// TIA Portal V19 export
FUNCTION_BLOCK "CameraConnectionTCP"   // FB2, LAD
{ S7_Optimized_Access := 'TRUE' }
// stored: MemoryReserve 100, SetENOAutomatically false
   VAR_INPUT
      Enable : Bool;
      Execute : Bool;
      Reset : Bool;
      ConnectionTimer : Time;
   END_VAR
   VAR_OUTPUT
      Status : "Status";
   END_VAR
   VAR_IN_OUT
      Parameters : TCON_IP_v4;
   END_VAR
   VAR
      TCON_Instance { ExternalAccessible := 'False'; ExternalVisible := 'False'; ExternalWritable := 'False'} : TCON;
      TDISCON_Instance { ExternalAccessible := 'False'; ExternalVisible := 'False'; ExternalWritable := 'False'} : TDISCON;
      TRCV_Instance { ExternalAccessible := 'False'; ExternalVisible := 'False'; ExternalWritable := 'False'} : TRCV;
      TSEND_Instance { ExternalAccessible := 'False'; ExternalVisible := 'False'; ExternalWritable := 'False'} : TSEND;
      Connection : Struct
         TCON : Struct
            REQ : Bool;
            BUSY : Bool;
            DONE : Bool;
            ERROR : Bool;
            STATUS : Word;
            CONNECTION_DATA : Struct
               InterfaceID : HW_ANY := 64;
               ID : HW_ANY := 1;
               ConnectionType : Byte := 16#0B;
               ActiveEstablished : Bool := false;
               RemodeAddress { S7_SetPoint := 'True'} : IP_V4;
               RemotePort : UInt;
               LocalPort : UInt := 2000;
            END_STRUCT;
         END_STRUCT;
         TDISCON : Struct
            REQ : Bool;
            BUSY : Bool;
            DONE : Bool;
            ERROR : Bool;
            STATUS : Word;
         END_STRUCT;
         TSEND : Struct
            REQ : Bool;
            LEN : UDInt;
            BUSY : Bool;
            DONE : Bool;
            ERROR : Bool;
            STATUS : Word;
         END_STRUCT;
         TRVC : Struct
            ENABLE : Bool;
            ADHOC : Bool := TRUE;
            LEN : UDInt;
            NDR : Bool;
            BUSY : Bool;
            RVC_LEN : UDInt;
            ERROR : Bool;
            STATUS : Word;
         END_STRUCT;
      END_STRUCT;
      Data : Struct
         RVC : Array[0..999] of Byte;
         SEND : Array[0..999] of Byte;
      END_STRUCT;
      State : "s_changeState";
      Timers : Struct
         WatchdogInit : "s_TON";
         WatchdogCamera : "s_TON";
         WatchdogInitRVC { S7_SetPoint := 'True'} : "s_TON";
         WatchdogMachineStart { S7_SetPoint := 'True'} : "s_TON";
      END_STRUCT;
      MessageGenerating : Struct
         i : Int;
         len : DInt;
         "string" : String[100];
         chars : Array[0..99] of Char;
      END_STRUCT;
      Local : Struct
         MessageSent : Bool;
         MessageSentCounter : SInt;
         prevState : Int;
      END_STRUCT;
      F_TRIG_Enable { ExternalAccessible := 'False'; ExternalVisible := 'False'; ExternalWritable := 'False'} : F_TRIG;
      R_TRIG_Execute { ExternalAccessible := 'False'; ExternalVisible := 'False'; ExternalWritable := 'False'} : R_TRIG;
      R_TRIG_Enable { ExternalAccessible := 'False'; ExternalVisible := 'False'; ExternalWritable := 'False'} : R_TRIG;
      Connected : Bool;
      DebugCounter : DInt;
   END_VAR
   VAR CONSTANT
      S_INITIALIZE : Int := 1;
      S_DISCONNECT : Int := 10;
      S_ERROR : Int := 20;
      S_ENABLE_RVC : Int := 30;
      S_MACHINE_START : Int := 40;
      S_IDLE : Int := 50;
      S_START_CAMERA : Int := 60;
      S_REPEAT : Int := 70;
      STATE_TEST : Int := 100;
      COMAND_SEND_MACHINE_START : String := 'command: machine_start';
      COMMAND_RVC_MACHINE_START : String := 'command: camera_ready';
      COMMAND_SEND_START_CONTROL : String := 'command: start_control';
      COMMAND_RVC_CONTROL_DONE : String := 'command: control_done';
      E_CONNECTION_TIMEOUT : Word := 16#8000;
      E_WRONG_RESPONSE_MACHINE_START : Word := 16#8001;
      E_START_MACHINE_NOT_SENT : Word := 16#8002;
      E_START_MACHINE_NO_RESPONSE : Word := 16#8003;
      E_WRONG_RESPONSE_CAMERA : Word := 16#8004;
      E_CAMERA_NO_RESPONSE : Word := 16#8005;
      E_CAMERA_NOT_SENT : Word := 16#8006;
      E_TRCV_ERROR : Word := 16#8007;
      E_TRCV_TIMEOUT : Word := 16#8008;
      E_TCON_ERROR : Word := 16#8009;
      E_TDISCON_ERROR : Word := 16#8010;
      E_TSEND_ERROR : Word := 16#8011;
   END_VAR
   // Connection.TCON.CONNECTION_DATA.RemodeAddress.ADDR[1] := 192;
   // Connection.TCON.CONNECTION_DATA.RemodeAddress.ADDR[2] := 168;
   // Connection.TCON.CONNECTION_DATA.RemodeAddress.ADDR[3] := 0;
   // Connection.TCON.CONNECTION_DATA.RemodeAddress.ADDR[4] := 69;
BEGIN

REGION Network 1 (SCL)
   //************************************************************
   //===Author: Mateusz Połojko
   //-----Linkedin: https://pl.linkedin.com/in/mateusz-po%C5%82ojko-52a3541b1
   //-----Github: https://github.com/Bhazel95
   //===Description:
   //-----Camera control via TCP/IP
   //===Customer:
   //-----Apator Powogaz S.A.
   //************************************************************
END_REGION

REGION Network 2
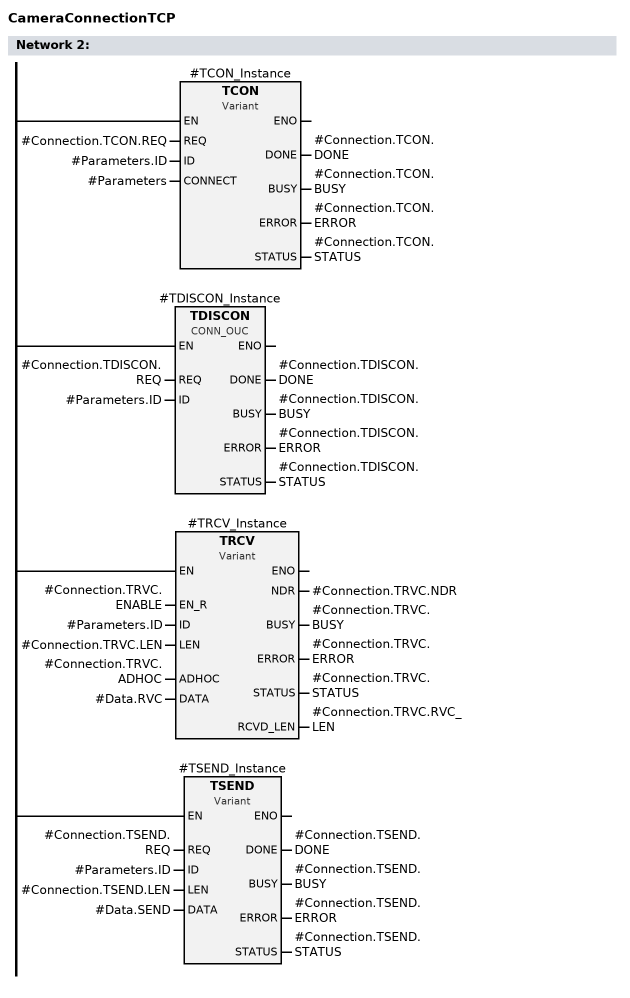
   RUNG wire#powerrail
      { S7_Templates := "[con_type := Variant, id_type := CONN_OUC]" } #TCON_Instance.TCON(REQ := #Connection.TCON.REQ, ID := #Parameters.ID, CONNECT := #Parameters, DONE => #Connection.TCON.DONE, BUSY => #Connection.TCON.BUSY, ERROR => #Connection.TCON.ERROR, STATUS => #Connection.TCON.STATUS)
   END_RUNG
   RUNG wire#powerrail
      { S7_Templates := "id_type := CONN_OUC" } #TDISCON_Instance.TDISCON(REQ := #Connection.TDISCON.REQ, ID := #Parameters.ID, DONE => #Connection.TDISCON.DONE, BUSY => #Connection.TDISCON.BUSY, ERROR => #Connection.TDISCON.ERROR, STATUS => #Connection.TDISCON.STATUS)
   END_RUNG
   RUNG wire#powerrail
      { S7_Templates := "[card := 1, ptr_type := Variant, value_type := UDInt, id_type := CONN_OUC]" } #TRCV_Instance.TRCV(EN_R := #Connection.TRVC.ENABLE, ID := #Parameters.ID, LEN := #Connection.TRVC.LEN, ADHOC := #Connection.TRVC.ADHOC, DATA := #Data.RVC, NDR => #Connection.TRVC.NDR, BUSY => #Connection.TRVC.BUSY, ERROR => #Connection.TRVC.ERROR, STATUS => #Connection.TRVC.STATUS, RCVD_LEN => #Connection.TRVC.RVC_LEN)
   END_RUNG
   RUNG wire#powerrail
      { S7_Templates := "[data_type := Variant, len_type := UDInt, id_type := CONN_OUC]" } #TSEND_Instance.TSEND(REQ := #Connection.TSEND.REQ, ID := #Parameters.ID, LEN := #Connection.TSEND.LEN, DATA := #Data.SEND, DONE => #Connection.TSEND.DONE, BUSY => #Connection.TSEND.BUSY, ERROR => #Connection.TSEND.ERROR, STATUS => #Connection.TSEND.STATUS)
   END_RUNG
   // the same network as SCL:
   #TCON_Instance(REQ := #Connection.TCON.REQ,   // TCON
                  ID := #Parameters.ID,
                  CONNECT := #Parameters,
                  DONE => #Connection.TCON.DONE,
                  BUSY => #Connection.TCON.BUSY,
                  ERROR => #Connection.TCON.ERROR,
                  STATUS => #Connection.TCON.STATUS);
   #TDISCON_Instance(REQ := #Connection.TDISCON.REQ,   // TDISCON
                     ID := #Parameters.ID,
                     DONE => #Connection.TDISCON.DONE,
                     BUSY => #Connection.TDISCON.BUSY,
                     ERROR => #Connection.TDISCON.ERROR,
                     STATUS => #Connection.TDISCON.STATUS);
   #TRCV_Instance(EN_R := #Connection.TRVC.ENABLE,   // TRCV
                  ID := #Parameters.ID,
                  LEN := #Connection.TRVC.LEN,
                  ADHOC := #Connection.TRVC.ADHOC,
                  DATA := #Data.RVC,
                  NDR => #Connection.TRVC.NDR,
                  BUSY => #Connection.TRVC.BUSY,
                  ERROR => #Connection.TRVC.ERROR,
                  STATUS => #Connection.TRVC.STATUS,
                  RCVD_LEN => #Connection.TRVC.RVC_LEN);
   #TSEND_Instance(REQ := #Connection.TSEND.REQ,   // TSEND
                   ID := #Parameters.ID,
                   LEN := #Connection.TSEND.LEN,
                   DATA := #Data.SEND,
                   DONE => #Connection.TSEND.DONE,
                   BUSY => #Connection.TSEND.BUSY,
                   ERROR => #Connection.TSEND.ERROR,
                   STATUS => #Connection.TSEND.STATUS);
END_REGION

REGION Network 3 (SCL)
   REGION TIMERS
       //WATCHDOG INICJALIZACJA POŁĄCZENIA
       #Timers.WatchdogInit.PT := #ConnectionTimer;
       #Timers.WatchdogInit.Timer(IN := #Timers.WatchdogInit.IN,
                                  PT := #Timers.WatchdogInit.PT);

       //WATCHDOG WYSYLANIE DANYCH DO ZROBIENIA ZDJĘCIA
       #Timers.WatchdogCamera.PT := T#5S;
       #Timers.WatchdogCamera.Timer(IN := #Timers.WatchdogCamera.IN,
                                    PT := #Timers.WatchdogCamera.PT);

       //WATCHDOG INICJALIZACJI POŁĄCZENIA
       #Timers.WatchdogInitRVC.PT := T#10S;
       #Timers.WatchdogInitRVC.Timer(IN := #Timers.WatchdogInitRVC.IN,
                                     PT := #Timers.WatchdogInitRVC.PT);

       //WATCHDOG MACHINE START
       #Timers.WatchdogMachineStart.PT := T#10S;
       #Timers.WatchdogMachineStart.Timer(IN := #Timers.WatchdogMachineStart.IN,
                                          PT := #Timers.WatchdogMachineStart.PT);
   END_REGION

   REGION R/F TRIG
       #F_TRIG_Enable(CLK:=#Enable);
       #R_TRIG_Execute(CLK:=#Execute);
       #R_TRIG_Enable(CLK:=#Enable);
   END_REGION


   CASE #State.state OF
       #S_INITIALIZE:
           //Funkcja wejścia
           IF #State.inputFlag AND NOT #State.outputFlag THEN
               #State.name := 'INICJALIZACJA POLACZENIA';
              // #State.name := 'ERROR';
               #Status.Busy := TRUE;
               #Status.Ready := FALSE;
               #Status.Done := FALSE;
               #Status.Error := FALSE;
               #Status.ErrorStatus := 16#0000;
               #Timers.WatchdogCamera.IN := FALSE;
               #Timers.WatchdogInit.IN := FALSE;
               #Timers.WatchdogInitRVC.IN := FALSE;
               #Timers.WatchdogMachineStart.IN := FALSE;
               #Connection.TRVC.ADHOC := TRUE;
               #Connection.TCON.REQ := TRUE;
               #Timers.WatchdogInit.IN := TRUE;
               #Connection.TCON.REQ := TRUE;
           END_IF;

           //Funkcja cykliczna
           IF NOT #State.inputFlag AND NOT #State.outputFlag THEN
               IF #Connection.TCON.STATUS = 16#0000 (* AND NOT #Connection.TCON.BUSY *) THEN
                   "changeState"(newState := #S_ENABLE_RVC,
                                 Data := #State);
               END_IF;

               IF #Timers.WatchdogInit.Timer.Q THEN
                   #Status.ErrorStatus  := #E_CONNECTION_TIMEOUT;
                   "changeState"(newState := #S_ERROR,
                                 Data := #State);
               END_IF;
           END_IF;

           //Funkcja wyjściowa 
           IF #State.outputFlag THEN
               #Timers.WatchdogInit.IN := FALSE;
           END_IF;

       #S_DISCONNECT:
           //Funkcja wejścia
           IF #State.inputFlag AND NOT #State.outputFlag THEN
               #State.name := 'DISCONNECT Z SIECIA';
               #Status.ErrorStatus  := 16#0000;
               #Connection.TCON.REQ := FALSE;
               #Connection.TSEND.REQ := FALSE;
               #Connection.TRVC.ENABLE := FALSE;
               #Connection.TDISCON.REQ := TRUE;
               #Status.ErrorStatus := 16#0000;
               #Timers.WatchdogCamera.IN := FALSE;
               #Timers.WatchdogInit.IN := FALSE;
               #Timers.WatchdogInitRVC.IN := FALSE;
               #Timers.WatchdogMachineStart.IN := FALSE;
               #Status.Error := FALSE;
           END_IF;

           //Funkcja cykliczna
           IF NOT #State.inputFlag AND NOT #State.outputFlag THEN
               IF NOT #Connection.TDISCON.BUSY AND NOT #Connection.TCON.BUSY THEN
                   #Connection.TDISCON.REQ := FALSE;
               END_IF;
               IF #Enable AND #Connection.TDISCON.REQ = FALSE  THEN
                   "changeState"(newState := #S_INITIALIZE,
                                 Data := #State);
               END_IF;
           END_IF;

           //Funkcja wyjściowa 
           IF #State.outputFlag THEN
               ;
           END_IF;

       #S_ERROR:
           //Funkcja wejścia
           IF #State.inputFlag AND NOT #State.outputFlag THEN
               #State.name := 'ERROR';
               #Status.Busy := FALSE;
               #Status.Ready := FALSE;
               #Status.Done := FALSE;
               #Status.Error := TRUE;
           END_IF;

           //Funkcja cykliczna
           IF NOT #State.inputFlag AND NOT #State.outputFlag THEN
               IF #Reset THEN
                   #Status.ErrorStatus  := 16#0000;
                   #Status.Error := FALSE;
                       "changeState"(newState := #S_DISCONNECT,
                                     Data := #State);
               END_IF;
           END_IF;

           //Funkcja wyjściowa 
           IF #State.outputFlag THEN
               ;
           END_IF;

       #S_ENABLE_RVC:
           //Funkcja wejścia
           IF #State.inputFlag AND NOT #State.outputFlag THEN
               #State.name := 'ZEZWOLENIE NA ODBIERANIE DANYCH';
               #Connection.TRVC.ADHOC := TRUE;
               #Timers.WatchdogInitRVC.IN := TRUE;
               #Connection.TRVC.ENABLE := TRUE;
           END_IF;

           //Funkcja cykliczna
           IF NOT #State.inputFlag AND NOT #State.outputFlag THEN
               IF #Connection.TRVC.STATUS = 16#7001 OR #Connection.TRVC.STATUS = 16#7002 THEN
                   "changeState"(newState := #S_MACHINE_START,
                                 Data := #State);
               END_IF;

               IF #Timers.WatchdogInitRVC.Timer.Q THEN
                   #Status.ErrorStatus  := #E_TRCV_TIMEOUT;
                   "changeState"(newState := #S_ERROR,
                                 Data := #State);
               END_IF;
           END_IF;

           //Funkcja wyjściowa 
           IF #State.outputFlag THEN
               #Timers.WatchdogInitRVC.IN := FALSE;
           END_IF;

       #S_MACHINE_START:
           //Funkcja wejścia
           IF #State.inputFlag AND NOT #State.outputFlag THEN
               #State.name := 'TWORZENIE WIADOMOSCI';
               #MessageGenerating.len := LEN(#COMAND_SEND_MACHINE_START);
               Strg_TO_Chars(Strg := #COMAND_SEND_MACHINE_START,
                             pChars := 0,
                             Cnt => #MessageGenerating.len,
                             Chars := #MessageGenerating.chars);
               FOR #MessageGenerating.i := 0 TO #MessageGenerating.len DO
                   #Data.SEND[#MessageGenerating.i] := CHAR_TO_BYTE(#MessageGenerating.chars[#MessageGenerating.i]);
               END_FOR;
               #Connection.TSEND.LEN := DINT_TO_UDINT(#MessageGenerating.len);
               #Timers.WatchdogMachineStart.IN := TRUE;
               #Local.MessageSent := FALSE; //ZMIENNA ODPOWIADAJĄCA ZA SPRAWDZENIE CZY WIADOMOŚĆ ZOSTAŁA WYSŁANA
               #State.name := 'OCZEKIWANIE NA DANE Z KAMERY';
               #Connection.TSEND.REQ := TRUE;
           END_IF;

           //Funkcja cykliczna
           IF NOT #State.inputFlag AND NOT #State.outputFlag THEN

               //WIADOMOŚĆ POMYŚLNIE WYSŁANA
               IF #Connection.TSEND.DONE THEN
                   #Local.MessageSent := TRUE;
               END_IF;

               //ODEBRANIE WIADOMOŚCI I DEKODOWANIE
               IF #Connection.TRVC.NDR AND #Local.MessageSent THEN
                   FOR #MessageGenerating.i := 0 TO UDINT_TO_INT(#Connection.TRVC.RVC_LEN) DO
                       #MessageGenerating.chars[#MessageGenerating.i] := BYTE_TO_CHAR(#Data.RVC[#MessageGenerating.i]);
                   END_FOR;
                   Chars_TO_Strg(Chars := #MessageGenerating.chars,
                                 pChars := 0,
                                 Cnt := UDINT_TO_UINT(#Connection.TRVC.RVC_LEN),
                                 Strg => #MessageGenerating.string);
                   IF #COMMAND_RVC_MACHINE_START = #MessageGenerating.string THEN
                       "changeState"(newState := #S_IDLE,
                                     Data := #State);
                   ELSIF #COMMAND_RVC_MACHINE_START <> #MessageGenerating.string THEN
                       #Status.ErrorStatus  := #E_WRONG_RESPONSE_MACHINE_START;
                       "changeState"(newState := #S_ERROR,
                                     Data := #State);
                   END_IF;
               END_IF;

               //TIMEOUT
               IF #Timers.WatchdogMachineStart.Timer.Q THEN
   (*                //JEŚLI JUŻ BYŁY 3 PRÓBY WYSŁANIA WIADOMOŚCI
                   IF #Local.MessageSentCounter > 3 THEN
                       IF NOT #Local.MessageSent THEN
                           #Status.ErrorStatus  := #E_START_MACHINE_NOT_SENT;
                       ELSIF #Local.MessageSent THEN
                           #Status.ErrorStatus  := #E_START_MACHINE_NO_RESPONSE;
                       END_IF;
                       "changeState"(newState := #S_ERROR,
                                     Data := #State);
                       //WYSYŁANIE WIADOMOŚCI DO 3 RAZY    
                   ELSE
                       #Local.MessageSentCounter := #Local.MessageSentCounter + 1;
                       #Local.prevState := #State.state;
                       "changeState"(newState := #S_REPEAT,
                                     Data := #State);
                   END_IF; *)
                   "changeState"(newState := #S_ERROR,
                                 Data := #State);
               END_IF;
           END_IF;

           //Funkcja wyjściowa 
           IF #State.outputFlag THEN
               #Connection.TSEND.REQ := FALSE;
               #Timers.WatchdogMachineStart.IN := FALSE;
           END_IF;

       #S_IDLE:
           //Funkcja wejścia
           IF #State.inputFlag AND NOT #State.outputFlag THEN
               #Local.MessageSentCounter := 0;
               #State.name := 'OCZEKIWANIE NA WODOMIERZ';
               #Status.Busy := FALSE;
               #Status.Ready := TRUE;
               //#Status.Done := FALSE;
               #Status.Error := FALSE;
           END_IF;

           //Funkcja cykliczna
           IF NOT #State.inputFlag AND NOT #State.outputFlag THEN
               IF #Execute THEN
                    "changeState"(newState := #S_START_CAMERA,
                                 Data := #State);
               END_IF;
           END_IF;

           //Funkcja wyjściowa 
           IF #State.outputFlag THEN
               #Status.Done := FALSE;
               #Status.Ready := FALSE;
               #Status.Busy := TRUE;
           END_IF;

       #S_START_CAMERA:
           //Funkcja wejścia
           IF #State.inputFlag AND NOT #State.outputFlag THEN
               #State.name := 'WYSYLANIE DANYCH';
               #Local.MessageSent := FALSE;
               #MessageGenerating.len := LEN(#COMMAND_SEND_START_CONTROL);
               Strg_TO_Chars(Strg := #COMMAND_SEND_START_CONTROL,
                             pChars := 0,
                             Cnt => #MessageGenerating.len,
                             Chars := #MessageGenerating.chars);
               FOR #MessageGenerating.i := 0 TO #MessageGenerating.len DO
                   #Data.SEND[#MessageGenerating.i] := CHAR_TO_BYTE(#MessageGenerating.chars[#MessageGenerating.i]);
               END_FOR;
               #State.name := 'OCZEKIWANIE NA DANE Z KAMERY';
               #Connection.TSEND.LEN := DINT_TO_UDINT(#MessageGenerating.len);
               #Timers.WatchdogCamera.IN := TRUE;
               #Connection.TSEND.REQ := TRUE;
           END_IF;

           //Funkcja cykliczna
           IF NOT #State.inputFlag AND NOT #State.outputFlag THEN
               //POTWIERDZENIE WYSŁANIA WIADOMOŚCI
               IF #Connection.TSEND.DONE THEN
                   #Local.MessageSent := TRUE;
               END_IF;

               //ODEBRANIE WIADOMOŚCI I DEKODOWANIE
               IF #Connection.TRVC.NDR AND #Local.MessageSent THEN
                   FOR #MessageGenerating.i := 0 TO UDINT_TO_INT(#Connection.TRVC.RVC_LEN) DO
                       #MessageGenerating.chars[#MessageGenerating.i] := BYTE_TO_CHAR(#Data.RVC[#MessageGenerating.i]);
                   END_FOR;
                   Chars_TO_Strg(Chars := #MessageGenerating.chars,
                                 pChars := 0,
                                 Cnt := UDINT_TO_UINT(#Connection.TRVC.RVC_LEN),
                                 Strg => #MessageGenerating.string);
                   IF #COMMAND_RVC_CONTROL_DONE = #MessageGenerating.string THEN
                       #Status.Done := TRUE;
                       #DebugCounter := #DebugCounter + 1;
                       "changeState"(newState := #S_IDLE,
                                     Data := #State);
                   ELSIF #COMMAND_RVC_CONTROL_DONE <> #MessageGenerating.string THEN
                       #Status.ErrorStatus := #E_WRONG_RESPONSE_CAMERA;
                       "changeState"(newState := #S_ERROR,
                                     Data := #State);
                   END_IF; 
                   //#Status.Done := TRUE;
                   "changeState"(newState := #S_IDLE,
                                 Data := #State);
               END_IF;

               //TIMEOUT
               IF #Timers.WatchdogCamera.Timer.Q THEN
   (*                //JEŚLI JUŻ BYŁY 3 PRÓBY WYSŁANIA WIADOMOŚCI
                   IF #Local.MessageSentCounter > 3 THEN
                       IF NOT #Local.MessageSent THEN
                           #Status.ErrorStatus := #E_CAMERA_NOT_SENT;
                       ELSIF #Local.MessageSent THEN
                           #Status.ErrorStatus := #E_CAMERA_NO_RESPONSE;
                       END_IF;
                       "changeState"(newState := #S_ERROR,
                                     Data := #State);
                       //WYSYŁANIE WIADOMOŚCI DO 3 RAZY    
                   ELSE
                       #Local.MessageSentCounter := #Local.MessageSentCounter + 1;
                       #Local.prevState := #State.state;
                       "changeState"(newState := #S_REPEAT,
                                     Data := #State);
                   END_IF; 
                   "changeState"(newState := #S_ERROR,
                                 Data := #State); *)
                   "changeState"(newState := #S_ERROR,
                                 Data := #State);
               END_IF;
           END_IF;

           //Funkcja wyjściowa 
           IF #State.outputFlag THEN
               #Connection.TSEND.REQ := FALSE;
               #Timers.WatchdogCamera.IN := FALSE;
           END_IF;

       #S_REPEAT:
           "changeState"(newState := #Local.prevState,
                         Data := #State);
           //TESTOWANIE    
       #STATE_TEST:
           ;

   END_CASE;

   //GLOBAL ERRORS
   IF #Connection.TCON.ERROR THEN
       #Status.ErrorStatus := #E_TCON_ERROR;
       "changeState"(newState := #S_ERROR,
                     Data := #State);
    ELSIF #Connection.TRVC.ERROR THEN
       #Status.ErrorStatus := #E_TRCV_ERROR;
       "changeState"(newState := #S_ERROR,
                     Data := #State); 
   ELSIF #Connection.TSEND.ERROR THEN
       #Status.ErrorStatus := #E_TSEND_ERROR;
       "changeState"(newState := #S_ERROR,
                     Data := #State);
   (* ELSIF #Connection.TDISCON.ERROR THEN
       #Status.ErrorStatus := #E_TDISCON_ERROR;
       "changeState"(newState := #S_ERROR,
                     Data := #State); *)
   END_IF;

   //DISABLE FUNCTION BLOCK
   IF  #F_TRIG_Enable.Q  THEN
       "changeState"(newState := #S_DISCONNECT,
                     Data := #State);
   END_IF;

   IF #R_TRIG_Enable.Q THEN
       "changeState"(newState := #S_INITIALIZE,
                     Data := #State);
   END_IF;

   REGION Change state
       IF #State.inputFlag AND NOT #State.outputFlag THEN
           #State.inputFlag := FALSE;
       END_IF;
       #State.outputFlag := FALSE;
   END_REGION
END_REGION
END_FUNCTION_BLOCK
